Staubli VAL3: stop.pgx

program stop()
  local num l_nI
begin
  putln("TaskStatus: "+toString("",taskStatus(sInputBuffering)))
  bInputBuffering=false
  bTaskManager=false
  resetMotion()
  //wait(taskStatus(sInputBuffering)==0)
  delay(2)
  if taskStatus(sInputBuffering)!=0
    taskKill(sInputBuffering)
  endIf
  putln("TaskStatus: "+toString("",taskStatus(sInputBuffering)))
  putln("Stopped.")
end
